Universal Robots PolyScope program: phoneAssemblyBucle.urp

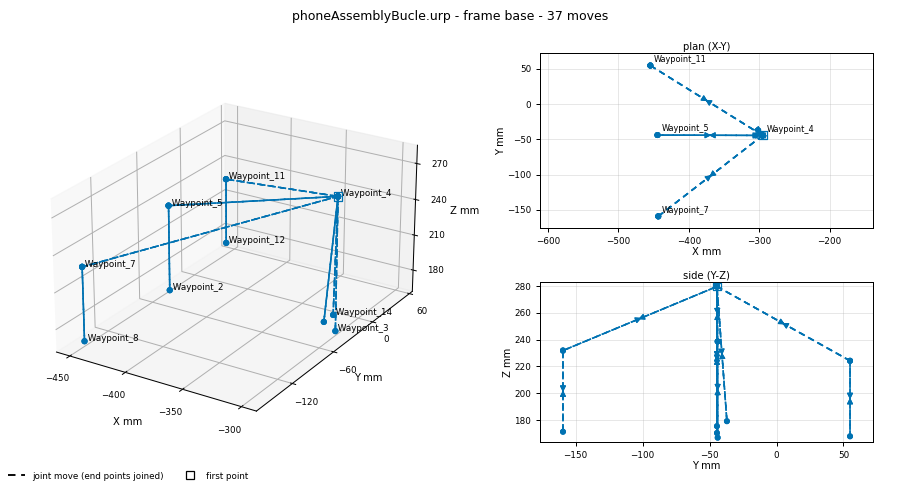
[picture p0: tool path of phoneAssemblyBucle.urp in frame base, 37 of 37 moves have a stored position in this frame; points joined in program order, loops and branches not executed]
Program phoneAssemblyBucle (installation=schmalz directory=/programs createdIn=5.2.0.61336 lastSavedIn=5.2.0.61336 robotSerialNumber=20185300040)
Calibrated DH parameters: a=[-0.000128, -0.221415, -0.194849, 0.000098, -0.000148, 0]; d=[0.152137, 33.879231, 13.968137, -47.716378, 0.085395, 0.092257]; alpha=[1.57105, 0.003021, -0.001826, 1.571145, -1.57192, 0]; deltaTheta=[0, 0.433042, -0.854582, 0.421536, 0.000002, 0]
Robot Program (runOnlyOnce=false)
  Set DigitalOutput pin=tool_out[0]; digitalValue=1
  'Base'
  MoveJ speed 60 deg/s, acceleration 80 deg/s^2 (useActiveTCP=true) feature=Base
    Waypoint Waypoint_4: TCP in base x=-295.068 y=-44.459 z=279.76 mm, rx=-1.7752 ry=-2.5817 rz=0.0079 rad; joints [-17.426, -97.252, 103.434, -96.793, -89.898, -38.552] deg
    Waypoint Waypoint_5: TCP in base x=-444.564 y=-43.95 z=238.725 mm, rx=-1.7752 ry=-2.5818 rz=0.0079 rad; joints [-11.405, -58.085, 65.864, -98.397, -89.864, -32.467] deg
    Waypoint Waypoint_2: TCP in base x=-444.562 y=-43.935 z=166.849 mm, rx=-1.7752 ry=-2.5819 rz=0.0079 rad; joints [-11.389, -53.13, 77.721, -115.207, -89.859, -32.47] deg
  Set DigitalOutput pin=tool_out[0]; digitalValue=0
  Set DigitalOutput pin=tool_out[1]; digitalValue=1
  Wait Sleep waitTime=0.3
  'Home'
  MoveJ speed 60 deg/s, acceleration 80 deg/s^2 (useActiveTCP=true) feature=Base
    Waypoint Waypoint_5: TCP in base x=-444.564 y=-43.95 z=238.725 mm, rx=-1.7752 ry=-2.5818 rz=0.0079 rad; joints [-11.405, -58.085, 65.864, -98.397, -89.864, -32.467] deg
    Waypoint Waypoint_4: TCP in base x=-295.068 y=-44.459 z=279.76 mm, rx=-1.7752 ry=-2.5817 rz=0.0079 rad; joints [-17.426, -97.252, 103.434, -96.793, -89.898, -38.552] deg
    Waypoint Waypoint_3: TCP in base x=-295.05 y=-44.472 z=170.342 mm, rx=-1.7751 ry=-2.5819 rz=0.0078 rad; joints [-17.402, -86.465, 125.272, -129.413, -89.872, -38.581] deg
  Set DigitalOutput pin=tool_out[1]; digitalValue=0
  Set DigitalOutput pin=tool_out[0]; digitalValue=1
  Wait Sleep waitTime=0.3
  'Battery'
  MoveJ speed 60 deg/s, acceleration 80 deg/s^2 (useActiveTCP=true) feature=Base
    Waypoint Waypoint_4: TCP in base x=-295.068 y=-44.459 z=279.76 mm, rx=-1.7752 ry=-2.5817 rz=0.0079 rad; joints [-17.426, -97.252, 103.434, -96.793, -89.898, -38.552] deg
    Waypoint Waypoint_7: TCP in base x=-443.495 y=-159.485 z=231.893 mm, rx=-1.7752 ry=-2.5819 rz=0.0079 rad; joints [3.656, -51.005, 55.904, -95.516, -89.998, -17.385] deg
    Waypoint Waypoint_8: TCP in base x=-443.502 y=-159.473 z=171.26 mm, rx=-1.7752 ry=-2.5818 rz=0.0079 rad; joints [3.672, -47.641, 66.646, -109.625, -90, -17.382] deg
  Set DigitalOutput pin=tool_out[0]; digitalValue=0
  Set DigitalOutput pin=tool_out[1]; digitalValue=1
  Wait Sleep waitTime=0.3
  'Home'
  MoveJ speed 60 deg/s, acceleration 80 deg/s^2 (useActiveTCP=true) feature=Base
    Waypoint Waypoint_7: TCP in base x=-443.495 y=-159.485 z=231.893 mm, rx=-1.7752 ry=-2.5819 rz=0.0079 rad; joints [3.656, -51.005, 55.904, -95.516, -89.998, -17.385] deg
    Waypoint Waypoint_4: TCP in base x=-295.068 y=-44.459 z=279.76 mm, rx=-1.7752 ry=-2.5817 rz=0.0079 rad; joints [-17.426, -97.252, 103.434, -96.793, -89.898, -38.552] deg
    Waypoint Waypoint_14: TCP in base x=-301.4 y=-37.043 z=179.139 mm, rx=-1.7752 ry=-2.5819 rz=0.0079 rad; joints [-18.489, -86.654, 122.505, -126.448, -89.858, -39.66] deg
  Set DigitalOutput pin=tool_out[1]; digitalValue=0
  Set DigitalOutput pin=tool_out[0]; digitalValue=1
  Wait Sleep waitTime=0.3
  'Top'
  MoveJ speed 60 deg/s, acceleration 80 deg/s^2 (useActiveTCP=true) feature=Base
    Waypoint Waypoint_4: TCP in base x=-295.068 y=-44.459 z=279.76 mm, rx=-1.7752 ry=-2.5817 rz=0.0079 rad; joints [-17.426, -97.252, 103.434, -96.793, -89.898, -38.552] deg
    Waypoint Waypoint_11: TCP in base x=-454.752 y=54.914 z=224.265 mm, rx=-1.7752 ry=-2.5818 rz=0.0079 rad; joints [-23.529, -54.493, 63.88, -99.979, -89.745, -44.584] deg
    Waypoint Waypoint_12: TCP in base x=-454.749 y=54.914 z=167.862 mm, rx=-1.7752 ry=-2.5818 rz=0.0079 rad; joints [-23.516, -50.598, 72.932, -112.924, -89.742, -44.583] deg
  Set DigitalOutput pin=tool_out[0]; digitalValue=0
  Set DigitalOutput pin=tool_out[1]; digitalValue=1
  Wait Sleep waitTime=0.3
  'Home'
  MoveJ speed 60 deg/s, acceleration 80 deg/s^2 (useActiveTCP=true) feature=Base
    Waypoint Waypoint_11: TCP in base x=-454.752 y=54.914 z=224.265 mm, rx=-1.7752 ry=-2.5818 rz=0.0079 rad; joints [-23.529, -54.493, 63.88, -99.979, -89.745, -44.584] deg
    Waypoint Waypoint_4: TCP in base x=-295.068 y=-44.459 z=279.76 mm, rx=-1.7752 ry=-2.5817 rz=0.0079 rad; joints [-17.426, -97.252, 103.434, -96.793, -89.898, -38.552] deg
    Waypoint Waypoint_13: TCP in base x=-305.088 y=-44.499 z=175.425 mm, rx=-1.7751 ry=-2.5818 rz=0.0079 rad; joints [-16.78, -84.895, 121.803, -127.519, -89.869, -37.951] deg
  Set DigitalOutput pin=tool_out[1]; digitalValue=0
  Set DigitalOutput pin=tool_out[0]; digitalValue=1
  Wait Sleep waitTime=0.3
  MoveJ speed 60 deg/s, acceleration 80 deg/s^2 (useActiveTCP=true) feature=Base
    Waypoint Waypoint_4: TCP in base x=-295.068 y=-44.459 z=279.76 mm, rx=-1.7752 ry=-2.5817 rz=0.0079 rad; joints [-17.426, -97.252, 103.434, -96.793, -89.898, -38.552] deg
  'Bucle'
  Wait Sleep waitTime=2
  'Home'
  MoveJ speed 60 deg/s, acceleration 80 deg/s^2 (useActiveTCP=true) feature=Base
    Waypoint Waypoint_13: TCP in base x=-305.088 y=-44.499 z=175.425 mm, rx=-1.7751 ry=-2.5818 rz=0.0079 rad; joints [-16.78, -84.895, 121.803, -127.519, -89.869, -37.951] deg
  Set DigitalOutput pin=tool_out[0]; digitalValue=0
  Set DigitalOutput pin=tool_out[1]; digitalValue=1
  Wait Sleep waitTime=0.3
  'Top'
  MoveJ speed 60 deg/s, acceleration 80 deg/s^2 (useActiveTCP=true) feature=Base
    Waypoint Waypoint_4: TCP in base x=-295.068 y=-44.459 z=279.76 mm, rx=-1.7752 ry=-2.5817 rz=0.0079 rad; joints [-17.426, -97.252, 103.434, -96.793, -89.898, -38.552] deg
    Waypoint Waypoint_11: TCP in base x=-454.752 y=54.914 z=224.265 mm, rx=-1.7752 ry=-2.5818 rz=0.0079 rad; joints [-23.529, -54.493, 63.88, -99.979, -89.745, -44.584] deg
    Waypoint Waypoint_12: TCP in base x=-454.749 y=54.914 z=167.862 mm, rx=-1.7752 ry=-2.5818 rz=0.0079 rad; joints [-23.516, -50.598, 72.932, -112.924, -89.742, -44.583] deg
  Set DigitalOutput pin=tool_out[1]; digitalValue=0
  Set DigitalOutput pin=tool_out[0]; digitalValue=1
  Wait Sleep waitTime=0.3
  'Home'
  MoveJ speed 60 deg/s, acceleration 80 deg/s^2 (useActiveTCP=true) feature=Base
    Waypoint Waypoint_11: TCP in base x=-454.752 y=54.914 z=224.265 mm, rx=-1.7752 ry=-2.5818 rz=0.0079 rad; joints [-23.529, -54.493, 63.88, -99.979, -89.745, -44.584] deg
    Waypoint Waypoint_4: TCP in base x=-295.068 y=-44.459 z=279.76 mm, rx=-1.7752 ry=-2.5817 rz=0.0079 rad; joints [-17.426, -97.252, 103.434, -96.793, -89.898, -38.552] deg
    Waypoint Waypoint_14: TCP in base x=-301.4 y=-37.043 z=179.139 mm, rx=-1.7752 ry=-2.5819 rz=0.0079 rad; joints [-18.489, -86.654, 122.505, -126.448, -89.858, -39.66] deg
  Set DigitalOutput pin=tool_out[0]; digitalValue=0
  Set DigitalOutput pin=tool_out[1]; digitalValue=1
  Wait Sleep waitTime=0.3
  MoveJ speed 60 deg/s, acceleration 80 deg/s^2 (useActiveTCP=true) feature=Base
    Waypoint Waypoint_4: TCP in base x=-295.068 y=-44.459 z=279.76 mm, rx=-1.7752 ry=-2.5817 rz=0.0079 rad; joints [-17.426, -97.252, 103.434, -96.793, -89.898, -38.552] deg
    Waypoint Waypoint_7: TCP in base x=-443.495 y=-159.485 z=231.893 mm, rx=-1.7752 ry=-2.5819 rz=0.0079 rad; joints [3.656, -51.005, 55.904, -95.516, -89.998, -17.385] deg
    Waypoint Waypoint_8: TCP in base x=-443.502 y=-159.473 z=171.26 mm, rx=-1.7752 ry=-2.5818 rz=0.0079 rad; joints [3.672, -47.641, 66.646, -109.625, -90, -17.382] deg
  Set DigitalOutput pin=tool_out[1]; digitalValue=0
  Set DigitalOutput pin=tool_out[0]; digitalValue=1
  Wait Sleep waitTime=0.3
  MoveJ speed 60 deg/s, acceleration 80 deg/s^2 (useActiveTCP=true) feature=Base
    Waypoint Waypoint_7: TCP in base x=-443.495 y=-159.485 z=231.893 mm, rx=-1.7752 ry=-2.5819 rz=0.0079 rad; joints [3.656, -51.005, 55.904, -95.516, -89.998, -17.385] deg
    Waypoint Waypoint_4: TCP in base x=-295.068 y=-44.459 z=279.76 mm, rx=-1.7752 ry=-2.5817 rz=0.0079 rad; joints [-17.426, -97.252, 103.434, -96.793, -89.898, -38.552] deg
    Waypoint Waypoint_3: TCP in base x=-295.05 y=-44.472 z=170.342 mm, rx=-1.7751 ry=-2.5819 rz=0.0078 rad; joints [-17.402, -86.465, 125.272, -129.413, -89.872, -38.581] deg
  Set DigitalOutput pin=tool_out[0]; digitalValue=0
  Set DigitalOutput pin=tool_out[1]; digitalValue=1
  Wait Sleep waitTime=0.3
  MoveJ speed 60 deg/s, acceleration 80 deg/s^2 (useActiveTCP=true) feature=Base
    Waypoint Waypoint_4: TCP in base x=-295.068 y=-44.459 z=279.76 mm, rx=-1.7752 ry=-2.5817 rz=0.0079 rad; joints [-17.426, -97.252, 103.434, -96.793, -89.898, -38.552] deg
    Waypoint Waypoint_5: TCP in base x=-444.564 y=-43.95 z=238.725 mm, rx=-1.7752 ry=-2.5818 rz=0.0079 rad; joints [-11.405, -58.085, 65.864, -98.397, -89.864, -32.467] deg
    Waypoint Waypoint_2: TCP in base x=-444.562 y=-43.935 z=166.849 mm, rx=-1.7752 ry=-2.5819 rz=0.0079 rad; joints [-11.389, -53.13, 77.721, -115.207, -89.859, -32.47] deg
  Set DigitalOutput pin=tool_out[1]; digitalValue=0
  Set DigitalOutput pin=tool_out[0]; digitalValue=1
  Wait Sleep waitTime=0.3
  MoveJ speed 60 deg/s, acceleration 80 deg/s^2 (useActiveTCP=true) feature=Base
    Waypoint Waypoint_5: TCP in base x=-444.564 y=-43.95 z=238.725 mm, rx=-1.7752 ry=-2.5818 rz=0.0079 rad; joints [-11.405, -58.085, 65.864, -98.397, -89.864, -32.467] deg
    Waypoint Waypoint_4: TCP in base x=-295.068 y=-44.459 z=279.76 mm, rx=-1.7752 ry=-2.5817 rz=0.0079 rad; joints [-17.426, -97.252, 103.434, -96.793, -89.898, -38.552] deg
